(*

.. <legal notes>

legal notes
=================
| SPDX-FileCopyrightText: © 2026 Oleksandr Tiutyk <trofimich@gmail.com>
| SPDX-License-Identifier: LGPL-3.0-only
| For details check: LGPL-3.0-only_

.. _LGPL-3.0-only: https://www.gnu.org/licenses/lgpl-3.0.en.html

.. </legal notes>

*)

INTERFACE IExceptionSeverityResolver EXTENDS IObject

METHOD GetSeverity : ERROR_SEVERITY
VAR_INPUT
	sourceException : IException;	
	catchPoint : STRING;
END_VAR
END_METHOD

END_INTERFACE

(* stored: Version 1.1.0.1
   Itf IExceptionSeverityResolver: Id {9dd4ebba-8c36-4f3a-be68-2612aa16ed4f}
   Method GetSeverity: Id {794f398a-186b-441a-b010-30479414113d} *)
